// TIA Portal V17 export
// export: Created 2023-05-04T15:49:35.2103582Z, ExportSetting None, DisplayName Totally Integrated Automation Portal, DisplayVersion V17 Update 4, DisplayName TIA Portal Openness, DisplayVersion V17 Update 4, DisplayName TIA Portal Version Control Interface, DisplayVersion V17, DisplayName STEP 7 Professional, DisplayVersion V17 Update 4, DisplayName STEP 7 Safety, DisplayVersion V17, DisplayName WinCC Advanced / Unified PC, DisplayVersion V17 Update 4
FUNCTION "FC_AIn" : Void   // FC1, LAD
TITLE = FC_AIn
{ S7_Optimized_Access := 'TRUE' }
// Analog Input
// stored: SetENOAutomatically false
BEGIN

REGION Network 1: DESCRIPTION
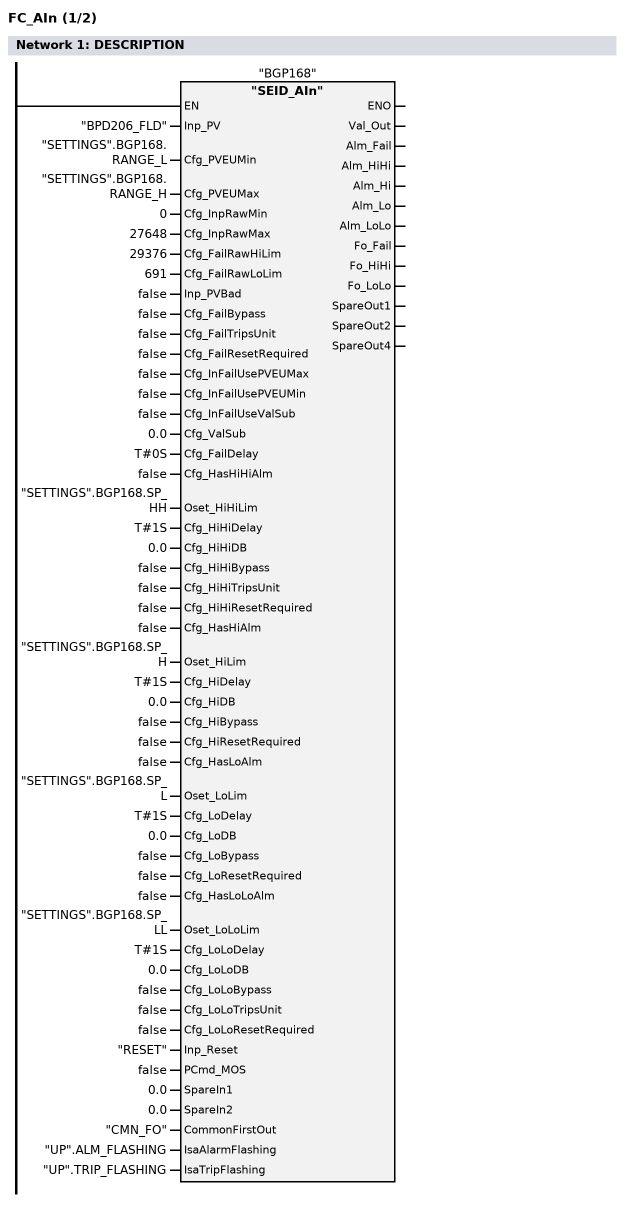
   RUNG wire#powerrail
      "BGP168"(Inp_PV := "BPD206_FLD", Cfg_PVEUMin := "SETTINGS".BGP168.RANGE_L, Cfg_PVEUMax := "SETTINGS".BGP168.RANGE_H, Cfg_InpRawMin := 0, Cfg_InpRawMax := 27648, Cfg_FailRawHiLim := 29376, Cfg_FailRawLoLim := 691, Inp_PVBad := false, Cfg_FailBypass := false, Cfg_FailTripsUnit := false, Cfg_FailResetRequired := false, Cfg_InFailUsePVEUMax := false, Cfg_InFailUsePVEUMin := false, Cfg_InFailUseValSub := false, Cfg_ValSub := 0.0, Cfg_FailDelay := T#0S, Cfg_HasHiHiAlm := false, Oset_HiHiLim := "SETTINGS".BGP168.SP_HH, Cfg_HiHiDelay := T#1S, Cfg_HiHiDB := 0.0, Cfg_HiHiBypass := false, Cfg_HiHiTripsUnit := false, Cfg_HiHiResetRequired := false, Cfg_HasHiAlm := false, Oset_HiLim := "SETTINGS".BGP168.SP_H, Cfg_HiDelay := T#1S, Cfg_HiDB := 0.0, Cfg_HiBypass := false, Cfg_HiResetRequired := false, Cfg_HasLoAlm := false, Oset_LoLim := "SETTINGS".BGP168.SP_L, Cfg_LoDelay := T#1S, Cfg_LoDB := 0.0, Cfg_LoBypass := false, Cfg_LoResetRequired := false, Cfg_HasLoLoAlm := false, Oset_LoLoLim := "SETTINGS".BGP168.SP_LL, Cfg_LoLoDelay := T#1S, Cfg_LoLoDB := 0.0, Cfg_LoLoBypass := false, Cfg_LoLoTripsUnit := false, Cfg_LoLoResetRequired := false, Inp_Reset := "RESET", PCmd_MOS := false, SpareIn1 := 0.0, SpareIn2 := 0.0, CommonFirstOut := "CMN_FO", IsaAlarmFlashing := "UP".ALM_FLASHING, IsaTripFlashing := "UP".TRIP_FLASHING, Val_Out =>, Alm_Fail =>, Alm_HiHi =>, Alm_Hi =>, Alm_Lo =>, Alm_LoLo =>, Fo_Fail =>, Fo_HiHi =>, Fo_LoLo =>, SpareOut1 =>, SpareOut2 =>, SpareOut4 =>)
   END_RUNG
   // the same network as SCL:
   "BGP168"(Inp_PV := "BPD206_FLD",   // "SEID_AIn"
            Cfg_PVEUMin := "SETTINGS".BGP168.RANGE_L,
            Cfg_PVEUMax := "SETTINGS".BGP168.RANGE_H,
            Cfg_InpRawMin := 0,
            Cfg_InpRawMax := 27648,
            Cfg_FailRawHiLim := 29376,
            Cfg_FailRawLoLim := 691,
            Inp_PVBad := false,
            Cfg_FailBypass := false,
            Cfg_FailTripsUnit := false,
            Cfg_FailResetRequired := false,
            Cfg_InFailUsePVEUMax := false,
            Cfg_InFailUsePVEUMin := false,
            Cfg_InFailUseValSub := false,
            Cfg_ValSub := 0.0,
            Cfg_FailDelay := T#0S,
            Cfg_HasHiHiAlm := false,
            Oset_HiHiLim := "SETTINGS".BGP168.SP_HH,
            Cfg_HiHiDelay := T#1S,
            Cfg_HiHiDB := 0.0,
            Cfg_HiHiBypass := false,
            Cfg_HiHiTripsUnit := false,
            Cfg_HiHiResetRequired := false,
            Cfg_HasHiAlm := false,
            Oset_HiLim := "SETTINGS".BGP168.SP_H,
            Cfg_HiDelay := T#1S,
            Cfg_HiDB := 0.0,
            Cfg_HiBypass := false,
            Cfg_HiResetRequired := false,
            Cfg_HasLoAlm := false,
            Oset_LoLim := "SETTINGS".BGP168.SP_L,
            Cfg_LoDelay := T#1S,
            Cfg_LoDB := 0.0,
            Cfg_LoBypass := false,
            Cfg_LoResetRequired := false,
            Cfg_HasLoLoAlm := false,
            Oset_LoLoLim := "SETTINGS".BGP168.SP_LL,
            Cfg_LoLoDelay := T#1S,
            Cfg_LoLoDB := 0.0,
            Cfg_LoLoBypass := false,
            Cfg_LoLoTripsUnit := false,
            Cfg_LoLoResetRequired := false,
            Inp_Reset := "RESET",
            PCmd_MOS := false,
            SpareIn1 := 0.0,
            SpareIn2 := 0.0,
            CommonFirstOut := "CMN_FO",
            IsaAlarmFlashing := "UP".ALM_FLASHING,
            IsaTripFlashing := "UP".TRIP_FLASHING);
END_REGION

REGION Network 2
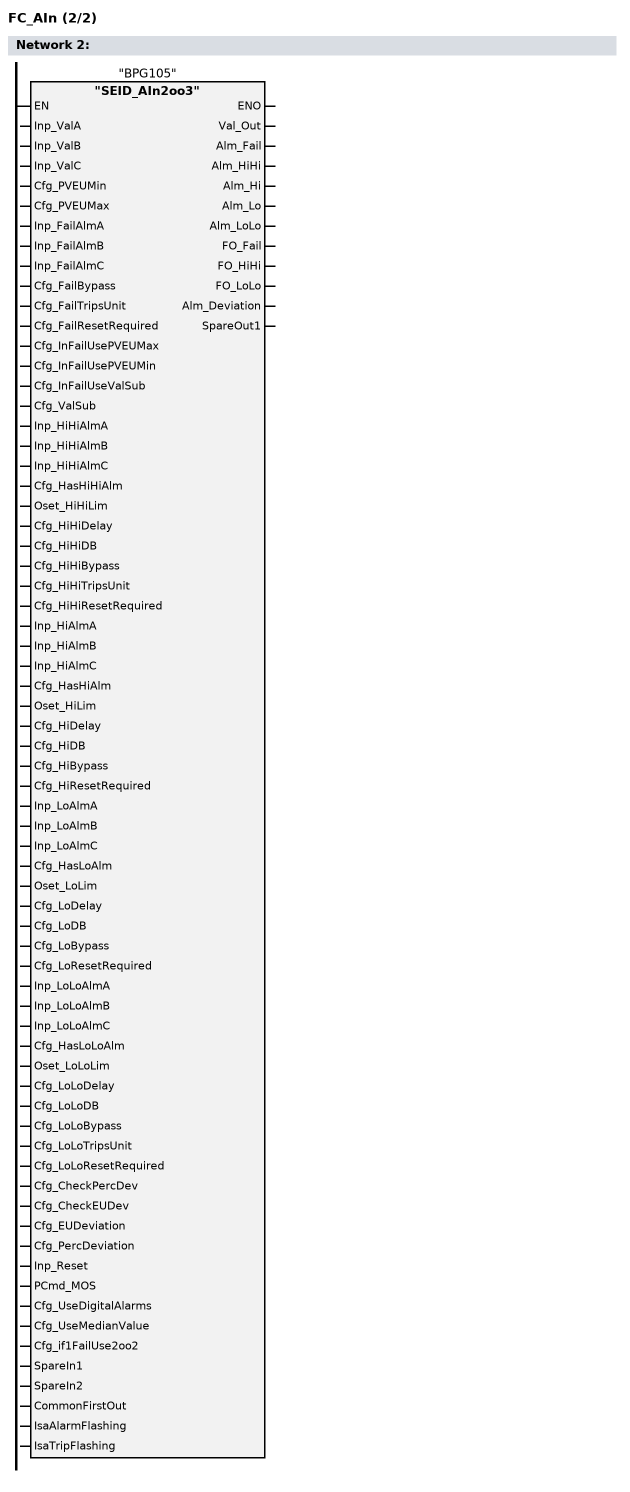
   RUNG wire#powerrail
      "BPG105"(Inp_ValA :=, Inp_ValB :=, Inp_ValC :=, Cfg_PVEUMin :=, Cfg_PVEUMax :=, Inp_FailAlmA :=, Inp_FailAlmB :=, Inp_FailAlmC :=, Cfg_FailBypass :=, Cfg_FailTripsUnit :=, Cfg_FailResetRequired :=, Cfg_InFailUsePVEUMax :=, Cfg_InFailUsePVEUMin :=, Cfg_InFailUseValSub :=, Cfg_ValSub :=, Inp_HiHiAlmA :=, Inp_HiHiAlmB :=, Inp_HiHiAlmC :=, Cfg_HasHiHiAlm :=, Oset_HiHiLim :=, Cfg_HiHiDelay :=, Cfg_HiHiDB :=, Cfg_HiHiBypass :=, Cfg_HiHiTripsUnit :=, Cfg_HiHiResetRequired :=, Inp_HiAlmA :=, Inp_HiAlmB :=, Inp_HiAlmC :=, Cfg_HasHiAlm :=, Oset_HiLim :=, Cfg_HiDelay :=, Cfg_HiDB :=, Cfg_HiBypass :=, Cfg_HiResetRequired :=, Inp_LoAlmA :=, Inp_LoAlmB :=, Inp_LoAlmC :=, Cfg_HasLoAlm :=, Oset_LoLim :=, Cfg_LoDelay :=, Cfg_LoDB :=, Cfg_LoBypass :=, Cfg_LoResetRequired :=, Inp_LoLoAlmA :=, Inp_LoLoAlmB :=, Inp_LoLoAlmC :=, Cfg_HasLoLoAlm :=, Oset_LoLoLim :=, Cfg_LoLoDelay :=, Cfg_LoLoDB :=, Cfg_LoLoBypass :=, Cfg_LoLoTripsUnit :=, Cfg_LoLoResetRequired :=, Cfg_CheckPercDev :=, Cfg_CheckEUDev :=, Cfg_EUDeviation :=, Cfg_PercDeviation :=, Inp_Reset :=, PCmd_MOS :=, Cfg_UseDigitalAlarms :=, Cfg_UseMedianValue :=, Cfg_if1FailUse2oo2 :=, SpareIn1 :=, SpareIn2 :=, CommonFirstOut :=, IsaAlarmFlashing :=, IsaTripFlashing :=, Val_Out =>, Alm_Fail =>, Alm_HiHi =>, Alm_Hi =>, Alm_Lo =>, Alm_LoLo =>, FO_Fail =>, FO_HiHi =>, FO_LoLo =>, Alm_Deviation =>, SpareOut1 =>)
   END_RUNG
   // the same network as SCL:
   "BPG105"();   // "SEID_AIn2oo3"
END_REGION
END_FUNCTION
